ABB RobotStudio station: Tema1_FINAL.rspag

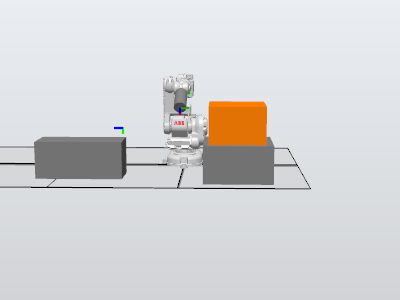
--- station ---
Station test_lab1 (saved by RobotStudio 23.2.10478.1)
Controller IRB140_6_81
  mechanical unit ROB_1: IRB140_6_81_C_03, 6 joints, base frame (0, 0, 0) mm
Layout (positions relative to the parent item):
  - IRB140_6_81_C_03 [mechanism, from %ABB.RobotStudio.Models.IRB140%\IRB140_6_81_C_G_03.rslib] at (0, 0, 0) mm; joint values [0, 0, 0, 0, 0.5236, 0] (rad or m)
  - CNC [part] at (351.33, 226.12, 300) mm, size 450 x 450 x 300 mm
  - masa [part] at (307.78, 183.15, 0) mm, size 550 x 550 x 300 mm
  - Conveyor [part] at (369.32, -1170.04, 0) mm, size 300 x 700 x 300 mm
  - Piesa [part] at (555.31, 275.89, 409.67) mm, rotated rx -90 ry 0 rz 0 deg, size 50 x 100 x 49.9 mm
  - MyNewTool [mechanism] at (506.29, 0, 679.5) mm, rotated rx 180 ry 60 rz 180 deg
      TCP MyNewTool at (0, 0, 200) mm
      links: Part_1
Attachment: MyNewTool is attached to IRB140_6_81_C_03 / Link6
EventTableEntry 2469: ActivationMode=2, Cyclic=false, Group=, Trigger=aa_gripper 2470, Actions=[EventTableActionAttach 2471], Comment=
EventTableTriggerIO 2470: Operator=0, IOValue=[1], IRC5Controller=? -1, SignalSource=IRB140_6_81 1186
EventTableActionAttach 2471: MountObject=true, FlangeIndext=0, FindNearest=true, AttachmentParent=MyNewTool 2631, AttachmentChild=? -1, Offset=[X=1, Y=0, Z=0, W=0, X=0, Y=1, Z=0, W=0, X=0, Y=0, Z=1, W=0, X=0, Y=0, Z=0, W=1]
EventTableEntry 2472: ActivationMode=2, Cyclic=false, Group=, Trigger=aa_gripper 2473, Actions=[EventTableActionDetach 2474], Comment=
EventTableTriggerIO 2473: Operator=0, IOValue=[0], IRC5Controller=? -1, SignalSource=IRB140_6_81 1186
EventTableActionDetach 2474: AttachmentParent=MyNewTool 2631, AttachmentChild=? -1

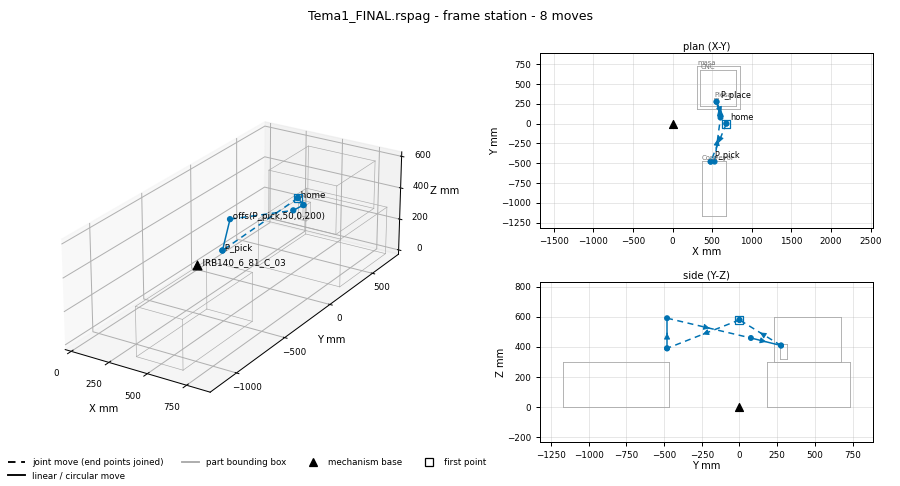
[picture p0: tool path of Tema1_FINAL.rspag in frame station, 8 of 8 moves have a stored position in this frame; points joined in program order, loops and branches not executed]
--- Controller Data/IRB140_6_81/RAPID/TASK1/PROGMOD/CalibData.mod ---
MODULE CalibData

    PERS tooldata MyNewTool:=[TRUE,[[0,0,200],[1,0,0,0]],[1,[0,0,1],[1,0,0,0],0,0,0]];
ENDMODULE

--- Controller Data/IRB140_6_81/RAPID/TASK1/PROGMOD/Module1.mod ---
MODULE Module1

        CONST robtarget home:=[[679.496774352,0,579.500016564],[0.500000024,0.000000013,0.86602539,0.000000007],[0,-1,0,0],[9E+09,9E+09,9E+09,9E+09,9E+09,9E+09]];
    CONST robtarget P_pick:=[[480.931,-479.942,390.985],[0,0,-0.707106781,0.707106781],[-1,0,-1,0],[9E+09,9E+09,9E+09,9E+09,9E+09,9E+09]];
    CONST robtarget P_place:=[[555.315,275.887,409.667],[0.707106781,-0.707106781,0,0],[0,0,0,0],[9E+09,9E+09,9E+09,9E+09,9E+09,9E+09]];
!
    ! Module:  Module1
    !
    ! Description:
    !   <Insert description here>
    !
    ! Author: Lenovo
    !
    ! Version: 1.0
    !
    !***********************************************************


    !***********************************************************
    !
    ! Procedure main
    !
    !   This is the entry point of your program
    !
    !***********************************************************
        PROC main()
        !Add your code here
        SetDO aa_gripper,0;
        MoveJ home,v1000,z100,MyNewTool\WObj:=wobj0;

        MoveJ offs(P_pick,0,0,0),v1000,fine,MyNewTool\WObj:=wobj0;
        MoveL P_pick,v1000,fine,MyNewTool\WObj:=wobj0;
        SetDO aa_gripper,1;
        WaitTime 0.5;
        MoveL offs(P_pick,50,0,200),v1000,fine,MyNewTool\WObj:=wobj0;

        MoveJ offs(P_place,50,-200,50),v1000,fine,MyNewTool\WObj:=wobj0;
        MoveL P_place,v1000,fine,MyNewTool\WObj:=wobj0;
        SetDO aa_gripper,0;
        WaitTime 0.5;
        MoveL offs(P_place,0,0,0),v1000,fine,MyNewTool\WObj:=wobj0;

        MoveJ home,v1000,z100,MyNewTool\WObj:=wobj0;
    ENDPROC
ENDMODULE

--- Controller Data/IRB140_6_81/SYSPAR/EIO.cfg ---
EIO:CFG_1.0:6:1::
#
EIO_SIGNAL:

      -Name "aa_gripper" -SignalType "DO" -Access "All"
